PROGRAM T03_xFAST
VAR
END_VAR

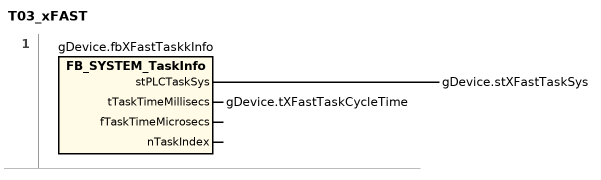
// NETWORK 1
gDevice.fbXFastTaskkInfo(tTaskTimeMillisecs => gDevice.tXFastTaskCycleTime); // FB_SYSTEM_TaskInfo
gDevice.stXFastTaskSys := gDevice.fbXFastTaskkInfo.stPLCTaskSys;

END_PROGRAM

(* stored: Version 1.1.0.1
   POU T03_xFAST: Id {ad4f51de-501d-4903-aced-fe727ff2695f}, SpecialFunc None *)
